FUNCTION F_MaxMarks : REAL
VAR_INPUT
	arr : ARRAY[1..10] OF REAL;
END_VAR
VAR_IN_OUT
    minMarks : REAL;
	maxMarks : REAL;
END_VAR
VAR
	i : INT;
END_VAR

minMarks := arr[1];
maxMarks := arr[1];

     FOR i:=2 TO 10 DO
		 IF arr[i] > maxMarks THEN
			 maxMarks := arr[i];
		 END_IF
		 
		 IF arr[i] < minMarks THEN
			  minMarks := arr[i];
		 END_IF
		 
	 END_FOR

END_FUNCTION

(* stored: Version 1.1.0.1, ProductVersion 3.1.4024.16
   POU F_MaxMarks: Id {434cf2c8-008f-45a4-960e-1be8bbde6103}, SpecialFunc None *)
